SYSTEM Test_FB
  (* Version 1.0, Author, 4DIAC-Consortium *)
  APPLICATION Fb_Test
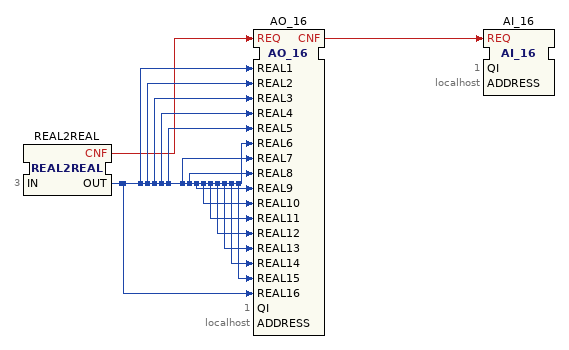
    FBS
      AO_16 : AO_16(QI := 1, ADDRESS := localhost);
      REAL2REAL : REAL2REAL(IN := 3);
      AI_16 : AI_16(QI := 1, ADDRESS := localhost);
    END_FBS
    EVENT_CONNECTIONS
      REAL2REAL.CNF TO AO_16.REQ;
      AO_16.CNF TO AI_16.REQ;
    END_CONNECTIONS
    DATA_CONNECTIONS
      REAL2REAL.OUT TO AO_16.REAL1;
      REAL2REAL.OUT TO AO_16.REAL2;
      REAL2REAL.OUT TO AO_16.REAL3;
      REAL2REAL.OUT TO AO_16.REAL4;
      REAL2REAL.OUT TO AO_16.REAL5;
      REAL2REAL.OUT TO AO_16.REAL6;
      REAL2REAL.OUT TO AO_16.REAL7;
      REAL2REAL.OUT TO AO_16.REAL8;
      REAL2REAL.OUT TO AO_16.REAL9;
      REAL2REAL.OUT TO AO_16.REAL10;
      REAL2REAL.OUT TO AO_16.REAL11;
      REAL2REAL.OUT TO AO_16.REAL12;
      REAL2REAL.OUT TO AO_16.REAL13;
      REAL2REAL.OUT TO AO_16.REAL14;
      REAL2REAL.OUT TO AO_16.REAL15;
      REAL2REAL.OUT TO AO_16.REAL16;
    END_CONNECTIONS
  END_APPLICATION
  APPLICATION UDP
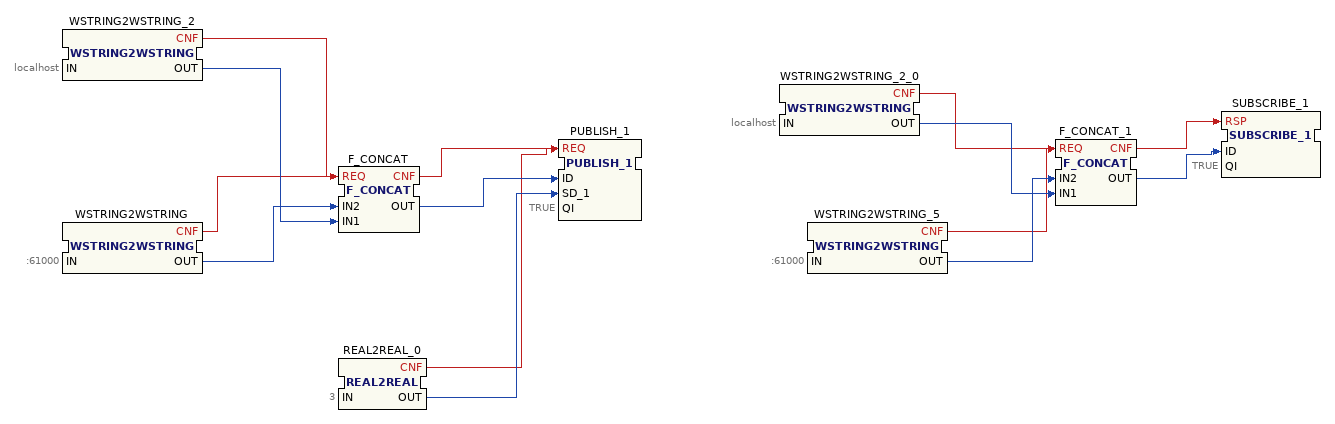
    FBS
      SUBSCRIBE_1 : SUBSCRIBE_1(QI := TRUE);
      PUBLISH_1 : PUBLISH_1(QI := TRUE);
      WSTRING2WSTRING : WSTRING2WSTRING(IN := :61000);
      F_CONCAT : F_CONCAT;
      WSTRING2WSTRING_2 : WSTRING2WSTRING(IN := localhost);
      F_CONCAT_1 : F_CONCAT;
      WSTRING2WSTRING_5 : WSTRING2WSTRING(IN := :61000);
      WSTRING2WSTRING_2_0 : WSTRING2WSTRING(IN := localhost);
      REAL2REAL_0 : REAL2REAL(IN := 3);
    END_FBS
    EVENT_CONNECTIONS
      WSTRING2WSTRING.CNF TO F_CONCAT.REQ;
      F_CONCAT.CNF TO PUBLISH_1.REQ;
      WSTRING2WSTRING_2.CNF TO F_CONCAT.REQ;
      WSTRING2WSTRING_2_0.CNF TO F_CONCAT_1.REQ;
      WSTRING2WSTRING_5.CNF TO F_CONCAT_1.REQ;
      F_CONCAT_1.CNF TO SUBSCRIBE_1.RSP;
      REAL2REAL_0.CNF TO PUBLISH_1.REQ;
    END_CONNECTIONS
    DATA_CONNECTIONS
      F_CONCAT.OUT TO PUBLISH_1.ID;
      WSTRING2WSTRING.OUT TO F_CONCAT.IN2;
      WSTRING2WSTRING_2.OUT TO F_CONCAT.IN1;
      WSTRING2WSTRING_5.OUT TO F_CONCAT_1.IN2;
      WSTRING2WSTRING_2_0.OUT TO F_CONCAT_1.IN1;
      F_CONCAT_1.OUT TO SUBSCRIBE_1.ID;
      REAL2REAL_0.OUT TO PUBLISH_1.SD_1;
    END_CONNECTIONS
  END_APPLICATION
  APPLICATION UDPPUBLISH
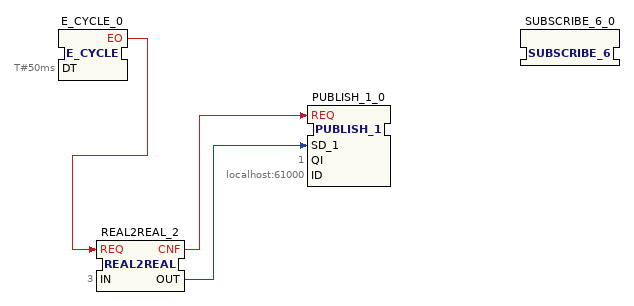
    FBS
      PUBLISH_1_0 : PUBLISH_1(QI := 1, ID := localhost:61000);
      REAL2REAL_2 : REAL2REAL(IN := 3);
      E_CYCLE_0 : E_CYCLE(DT := T#50ms);
      SUBSCRIBE_6_0 : SUBSCRIBE_6;
    END_FBS
    EVENT_CONNECTIONS
      REAL2REAL_2.CNF TO PUBLISH_1_0.REQ;
      E_CYCLE_0.EO TO REAL2REAL_2.REQ;
    END_CONNECTIONS
    DATA_CONNECTIONS
      REAL2REAL_2.OUT TO PUBLISH_1_0.SD_1;
    END_CONNECTIONS
  END_APPLICATION
  APPLICATION UDPSUBSCRIBE
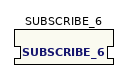
    FBS
      SUBSCRIBE_6 : SUBSCRIBE_6;
    END_FBS
  END_APPLICATION
  DEVICE FORTE_PC : FORTE_PC(MGR_ID := "localhost:61499")
    {SET_ATTRIBUTE(Profile, HOLOBLOC)}
    RESOURCE EMB_RES : EMB_RES
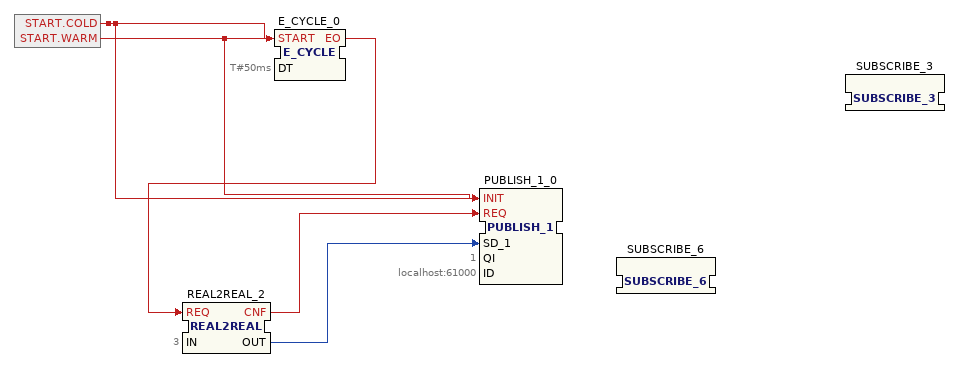
      FBS
        PUBLISH_1_0 : PUBLISH_1(QI := 1, ID := localhost:61000);
        REAL2REAL_2 : REAL2REAL(IN := 3);
        E_CYCLE_0 : E_CYCLE(DT := T#50ms);
        SUBSCRIBE_3 : SUBSCRIBE_3;
        SUBSCRIBE_6 : SUBSCRIBE_6;
      END_FBS
      EVENT_CONNECTIONS
        START.COLD TO PUBLISH_1_0.INIT;
        START.WARM TO PUBLISH_1_0.INIT;
        REAL2REAL_2.CNF TO PUBLISH_1_0.REQ;
        E_CYCLE_0.EO TO REAL2REAL_2.REQ;
        START.COLD TO E_CYCLE_0.START;
        START.WARM TO E_CYCLE_0.START;
      END_CONNECTIONS
      DATA_CONNECTIONS
        REAL2REAL_2.OUT TO PUBLISH_1_0.SD_1;
      END_CONNECTIONS
    END_RESOURCE
  END_DEVICE
  MAPPINGS
    UDPPUBLISH.PUBLISH_1_0 ON FORTE_PC.EMB_RES.PUBLISH_1_0;
    UDPPUBLISH.REAL2REAL_2 ON FORTE_PC.EMB_RES.REAL2REAL_2;
    UDPPUBLISH.E_CYCLE_0 ON FORTE_PC.EMB_RES.E_CYCLE_0;
    UDPSUBSCRIBE.SUBSCRIBE_6 ON FORTE_PC.EMB_RES.SUBSCRIBE_6;
  END_MAPPINGS
  SEGMENTS
    Ethernet : Ethernet;
  END_SEGMENTS
  LINKS
    FORTE_PC => Ethernet;
  END_LINKS
END_SYSTEM
